FUNCTION_BLOCK ENERGY_MODEL
  {SET_ATTRIBUTE(OpcUa, SERVICE)}
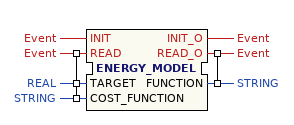
  EVENT_INPUT
    INIT;
    READ WITH COST_FUNCTION, TARGET;
  END_EVENT
  EVENT_OUTPUT
    INIT_O;
    READ_O WITH FUNCTION;
  END_EVENT
  VAR_INPUT
    TARGET : REAL; {SET_ATTRIBUTE(OpcUa, Constant)}
    COST_FUNCTION : STRING; {SET_ATTRIBUTE(OpcUa, Variable)}
  END_VAR
  VAR_OUTPUT
    FUNCTION : STRING; {SET_ATTRIBUTE(OpcUa, Variable)}
  END_VAR
END_FUNCTION_BLOCK
